# EPICS autosave request: iocBoot/generic_motors_ioc/dbSave/bluiceHutch.req
$(P)attenuation
$(P)beamsize_v
$(P)beamsize_h
$(P)beamsizeOption

$(P)px2mm_v_lo.A
$(P)px2mm_v_lo.B
$(P)px2mm_v_lo.C
$(P)px2mm_v_lo.D
$(P)px2mm_v_lo.CALC

$(P)px2mm_h_lo.A
$(P)px2mm_h_lo.B
$(P)px2mm_h_lo.C
$(P)px2mm_h_lo.D
$(P)px2mm_h_lo.CALC

$(P)px2mm_v_hi.A
$(P)px2mm_v_hi.B
$(P)px2mm_v_hi.C
$(P)px2mm_v_hi.D
$(P)px2mm_v_hi.CALC

$(P)px2mm_h_hi.A
$(P)px2mm_h_hi.B
$(P)px2mm_h_hi.C
$(P)px2mm_h_hi.D
$(P)px2mm_h_hi.CALC
